// TwinCAT 3 PLC project DAS_A2
// ProgramVersion: 3.1.4020.4
// libraries:
//   Tc2_Standard, * (Beckhoff Automation GmbH)
//   Tc2_System, * (Beckhoff Automation GmbH)
//   Tc3_Module, * (Beckhoff Automation GmbH)
// project tree:
//   DUTs/ ST_PALLET.TcDUT
//   / GlobalTextList.TcGTLO, PlcTask.TcTTO, Visualization Manager.TcVMO (not stored)
//   POUs/ MAIN.TcPOU
//   VISUs/ Visualization.TcVIS

CONFIGURATION DAS_A2
    RESOURCE PLC ON TwinCAT3
        TASK PlcTask(INTERVAL := T#10ms, PRIORITY := 20);
        PROGRAM MAIN WITH PlcTask : MAIN;
    END_RESOURCE
END_CONFIGURATION

// ---- DUTs/ST_PALLET.TcDUT
TYPE ST_PALLET :
STRUCT
	WS1: BOOL;
	WS2: BOOL;
	WS3: BOOL;
	STATE: INT := -1 ;
END_STRUCT
END_TYPE

// ---- POUs/MAIN.TcPOU
PROGRAM MAIN
VAR
	L1: BOOL;   //lock sesnsor1
	L2: BOOL;   //lock sesnsor2
	L3: BOOL;   //lock sesnsor3
	S1: BOOL;   //stopper1 
	S2: BOOL;   //stopper2
	S3: BOOL;   //stopper3
	BA1: BOOL;  //board available1
	BA2: BOOL;  //board available2
	BA3: BOOL;  //board available3
	P1: BOOL;   //presence sesnsor1
	P2: BOOL;   //presence sesnsor2
	P3: BOOL;   //presence sesnsor3
	T1: TON;    //timer for work station1
	T2: TON;    //timer for work station2
	T3: TON;    //timer for work station3
	COUNT_IN: INT;  //number of imported pallets 
	COUNT_OUT: INT;  //number of exported pallets
	PALLETI: ARRAY [1..10] OF ST_PALLET; //each index of this array use for one pallet
	PALLETV: ARRAY[1..10] OF ST_PALLET;  //for saving data of palleti array
	I: INT:=0;  //variable of for loop
	INPUT_PALLET: BOOL; //button for importing pallet to conveyor
	INPUT_PALLET_Pressed: BOOL; // these 3 input pallet used for counting input pallet button just one time in several cycle
	INPUT_PALLET_Released: BOOL;  //
	INPUT_PALLET_PressedBefore: BOOL;  //
	StartStop: BOOL;  //using for start and stop system
	MOTOR: BOOL; //motor of conveyor
	RESET_OUTV1: BOOL;  //exit pallet1 from system
	RESET_OUTV2: BOOL;  //exit pallet2 from system
	RESET_OUTV3: BOOL;  //exit pallet3 from system
	RESET_OUTV4: BOOL;  //exit pallet4 from system
	RESET_OUTV5: BOOL;  //exit pallet5 from system
	RESET_OUTV6: BOOL;  //exit pallet6 from system
	RESET_OUTV7: BOOL;  //exit pallet7 from system
	RESET_OUTV8: BOOL;  //exit pallet8 from system
	RESET_OUTV9: BOOL;  //exit pallet9 from system
	RESET_OUTV10: BOOL;  //exit pallet10 from system
END_VAR

T1(IN:=L1,PT:=T#5S);
T2(IN:=L2,PT:=T#5S);
T3(IN:=L3,PT:=T#5S);

IF INPUT_PALLET_Pressed THEN
	INPUT_PALLET_PressedBefore := TRUE;
ELSIF INPUT_PALLET_Pressed = FALSE AND INPUT_PALLET_PressedBefore THEN
	INPUT_PALLET := TRUE;
	INPUT_PALLET_PressedBefore := FALSE;
END_IF

//START AND INSERT PALLET TO THE SYSTEM AND FOR LOOP IS FOR PREVENTING PROGRAM FROM OVERWRITING DATA OF PALLETS ON PREVIOUS ARRAY INDEXES
	IF StartStop THEN
		MOTOR:=TRUE;
		IF INPUT_PALLET AND (COUNT_IN-COUNT_OUT)<11 THEN
		COUNT_IN:=COUNT_IN +1;
		FOR I:= 1 TO 10 DO
			IF PALLETI[I].STATE = -1 THEN
				PALLETI[I].STATE := 0;
				EXIT;
			END_IF
		END_FOR
		INPUT_PALLET := FALSE;
	END_IF
	
	
	//RESETING OUTPUT MEMORY FOR EACH PALLET
	IF RESET_OUTV1 THEN
			PALLETV[1].WS1:=FALSE;
			PALLETV[1].WS2:=FALSE;
			PALLETV[1].WS3:=FALSE;
			PALLETV[1].STATE:=0;
		END_IF
		IF RESET_OUTV2 THEN
			PALLETV[2].WS1:=FALSE;
			PALLETV[2].WS2:=FALSE;
			PALLETV[2].WS3:=FALSE;
			PALLETV[2].STATE:=0;
		END_IF
		IF RESET_OUTV3 THEN
			PALLETV[3].WS1:=FALSE;
			PALLETV[3].WS2:=FALSE;
			PALLETV[3].WS3:=FALSE;
			PALLETV[3].STATE:=0;
		END_IF
		IF RESET_OUTV4 THEN
			PALLETV[4].WS1:=FALSE;
			PALLETV[4].WS2:=FALSE;
			PALLETV[4].WS3:=FALSE;
			PALLETV[4].STATE:=0;
		END_IF
		IF RESET_OUTV5 THEN
			PALLETV[5].WS1:=FALSE;
			PALLETV[5].WS2:=FALSE;
			PALLETV[5].WS3:=FALSE;
			PALLETV[5].STATE:=0;
		END_IF
		IF RESET_OUTV6 THEN
			PALLETV[6].WS1:=FALSE;
			PALLETV[6].WS2:=FALSE;
			PALLETV[6].WS3:=FALSE;
			PALLETV[6].STATE:=0;
		END_IF
		IF RESET_OUTV7 THEN
			PALLETV[7].WS1:=FALSE;
			PALLETV[7].WS2:=FALSE;
			PALLETV[7].WS3:=FALSE;
			PALLETV[7].STATE:=0;
		END_IF
		IF RESET_OUTV8 THEN
			PALLETV[8].WS1:=FALSE;
			PALLETV[8].WS2:=FALSE;
			PALLETV[8].WS3:=FALSE;
			PALLETV[8].STATE:=0;
		END_IF
		IF RESET_OUTV9 THEN
			PALLETV[9].WS1:=FALSE;
			PALLETV[9].WS2:=FALSE;
			PALLETV[9].WS3:=FALSE;
			PALLETV[9].STATE:=0;
		END_IF
		IF RESET_OUTV10 THEN
			PALLETV[10].WS1:=FALSE;
			PALLETV[10].WS2:=FALSE;
			PALLETV[10].WS3:=FALSE;
			PALLETV[10].STATE:=0;
		END_IF
		
//MAIN FOR LOOP FOR WORKING ON PALLETS		
	FOR I:=1 TO 10 DO
		CASE PALLETI[I].STATE OF        //CHECKING DIFFERENT STATES FOR EACH PALLET
		   -1:
				CONTINUE;
			0:
			IF PALLETI[I].WS1 AND PALLETI[I].WS2 AND PALLETI[I].WS3 THEN
			    PALLETI[I].STATE:=10;
			END_IF	
			IF NOT L1 AND NOT L2 AND NOT L3 THEN
				IF NOT PALLETI[I].WS1 THEN
				PALLETI[I].STATE:=1;
				ELSIF NOT PALLETI[I].WS2 THEN
					PALLETI[I].STATE:=4;
				ELSIF NOT PALLETI[I].WS3 THEN
					PALLETI[I].STATE:=7;
				END_IF
			ELSIF L1 AND NOT L2 AND NOT L3 THEN
				IF NOT PALLETI[I].WS2 THEN
				PALLETI[I].STATE:=4;
				ELSIF NOT PALLETI[I].WS3 THEN
					PALLETI[I].STATE:=7;
				END_IF
			ELSIF L1 AND NOT L2 AND L3 THEN
				IF NOT PALLETI[I].WS2 THEN
				PALLETI[I].STATE:=4;
				END_IF
			ELSIF L1 AND L2 AND NOT L3 THEN
				IF NOT PALLETI[I].WS3 THEN
				PALLETI[I].STATE:=7;
				END_IF
			ELSIF NOT L1 AND L2 AND L3 THEN
				IF NOT PALLETI[I].WS1 THEN
				PALLETI[I].STATE:=1;
				END_IF
			ELSIF NOT L1 AND L2 AND NOT L3 THEN
				IF NOT PALLETI[I].WS3 THEN
				PALLETI[I].STATE:=7;
				END_IF
			ELSIF NOT L1 AND NOT L2 AND L3 THEN
				IF NOT PALLETI[I].WS1 THEN
					PALLETI[I].STATE:=1;
				ELSIF NOT PALLETI[I].WS2 THEN
					PALLETI[I].STATE:=4;
				END_IF
			END_IF
		
			1:  //WORK STATION1 WORKS ON PALLET UP TO STATE3
			IF PALLETI[I].WS1 AND PALLETI[I].WS2 AND PALLETI[I].WS3 THEN
			    PALLETI[I].STATE:=10;
			ELSIF NOT PALLETI[I].WS1 THEN
				IF NOT L1 AND P1 THEN
				BA1:=TRUE;
                S1:=TRUE;
				PALLETI[I].STATE:=2;
			    END_IF
			END_IF
			
			2:
			IF L1 THEN
				T1(IN:=L1,PT:=T#5S);
			    BA1:=FALSE;
			    S1:=FALSE;
				IF T1.Q THEN
					PALLETI[I].STATE:=3;
				END_IF
			END_IF
			
            3:
			IF NOT L1 THEN
				PALLETI[I].WS1:=1;
				IF PALLETI[I].WS1 AND PALLETI[I].WS2 AND PALLETI[I].WS3 THEN
			    PALLETI[I].STATE:=10;
				END_IF
				PALLETI[I].STATE:=0;
			END_IF

			4:   //WORK STATION2 WORKS ON PALLET UP TO STATE7
			IF PALLETI[I].WS1 AND PALLETI[I].WS2 AND PALLETI[I].WS3 THEN
			    PALLETI[I].STATE:=10;
			ELSIF NOT PALLETI[I].WS2 THEN
				IF NOT L2 AND P2 THEN
				BA2:=TRUE;
				S2:=TRUE;
				PALLETI[I].STATE:=5;
			    END_IF
			END_IF
			
            5:
			IF L2 THEN
				BA2:=FALSE;
			    S2:=FALSE;
				IF T2.Q THEN
					PALLETI[I].STATE:=6;
			    END_IF
			END_IF
			
			6:
			IF NOT L2 THEN
				PALLETI[I].WS2:=1;
				IF PALLETI[I].WS1 AND PALLETI[I].WS2 AND PALLETI[I].WS3 THEN
			    PALLETI[I].STATE:=10;
				END_IF
				PALLETI[I].STATE:=0;
			END_IF
			
			7:   //WORK STATION3 WORKS ON PALLET UP TO STATE9
			IF PALLETI[I].WS1 AND PALLETI[I].WS2 AND PALLETI[I].WS3 THEN
			    PALLETI[I].STATE:=10;
			ELSIF NOT PALLETI[I].WS3 THEN
				IF NOT L3 AND P3 THEN
				BA3:=TRUE;
				S3:=TRUE;
				PALLETI[I].STATE:=8;
			    END_IF
			END_IF
			
			8:
			IF L3 THEN
				BA3:=FALSE;
			    S3:=FALSE;
			    IF T3.Q THEN
					PALLETI[I].STATE:=9;
				END_IF
			END_IF
			
			9:
			IF NOT L3 THEN
				PALLETI[I].WS3:=1;
				IF PALLETI[I].WS1 AND PALLETI[I].WS2 AND PALLETI[I].WS3 THEN
			    PALLETI[I].STATE:=10;
				END_IF
				PALLETI[I].STATE:=0;
			END_IF
			
			10:    //TRANSFERING DATA OF PALLETI TO PALLETV AND RESET THE PALLET AND TURN IT BACK
				
				IF  PALLETI[I].WS1 AND PALLETI[I].WS2 AND PALLETI[I].WS3 THEN
					PALLETV[I].WS1:=PALLETI[I].WS1;
					PALLETV[I].WS2:=PALLETI[I].WS2;
					PALLETV[I].WS3:=PALLETI[I].WS3;
					PALLETV[I].STATE:=PALLETI[I].STATE;
			
				
				END_IF
				PALLETI[I].WS1:=FALSE;
				PALLETI[I].WS2:=FALSE;
				PALLETI[I].WS3:=FALSE;
				PALLETI[I].STATE:=-1;
				COUNT_OUT:=COUNT_OUT+1;
		
		END_CASE
	END_FOR
	ELSE 
		MOTOR:=FALSE;
END_IF

END_PROGRAM

// ---- GlobalTextList.TcGTLO
TEXTLIST GlobalTextList
  10 = 'BA1'
  9 = 'BA2'
  11 = 'BA3'
  41 = 'EXIT PALLET1'
  50 = 'EXIT PALLET10'
  42 = 'EXIT PALLET2'
  43 = 'EXIT PALLET3'
  44 = 'EXIT PALLET4'
  45 = 'EXIT PALLET5'
  46 = 'EXIT PALLET6'
  47 = 'EXIT PALLET7'
  48 = 'EXIT PALLET8'
  49 = 'EXIT PALLET9'
  18 = 'Input Pallet'
  3 = 'L1'
  4 = 'L2'
  5 = 'L3'
  15 = 'Motor'
  6 = 'P1'
  7 = 'P2'
  8 = 'P3'
  19 = 'Pallet 1'
  28 = 'Pallet 10'
  20 = 'Pallet 2'
  21 = 'Pallet 3'
  22 = 'Pallet 4'
  23 = 'Pallet 5'
  24 = 'Pallet 6'
  25 = 'Pallet 7'
  26 = 'Pallet 8'
  27 = 'Pallet 9'
  31 = 'R'
  30 = 'RESET PALLET1'
  40 = 'RESET PALLET10'
  32 = 'RESET PALLET2'
  33 = 'RESET PALLET3'
  34 = 'RESET PALLET4'
  35 = 'RESET PALLET5'
  36 = 'RESET PALLET6'
  37 = 'RESET PALLET7'
  38 = 'RESET PALLET8'
  39 = 'RESET PALLET9'
  17 = 'Start'
  29 = 'StartStop'
  16 = 'Stop'
  12 = 'Stopper1'
  13 = 'Stopper2'
  14 = 'Stopper3'
  1 = 'WS1'
  2 = 'WS2'
  0 = 'WS3'
END_TEXTLIST

// ---- VISUs/Visualization.TcVIS
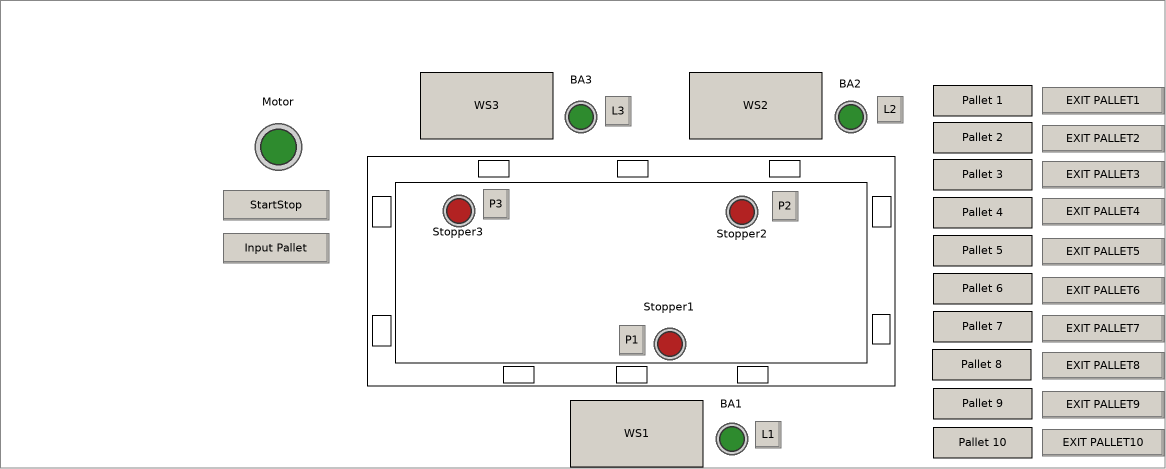
VISUALIZATION Visualization  // 1166x469
    RoundedRectangle (367,156 528x230)
    RoundedRectangle (395,182 472x181)
    Rectangle (570,400 133x67), "WS1", colour toggle: MAIN.T1.Q
    Rectangle (420,72 133x67), "WS3", colour toggle: MAIN.T3.Q
    Rectangle (689,72 133x67), "WS2", colour toggle: MAIN.T2.Q
    Button (755,421 26x27), "L1", text variable: MAIN.L1, colour toggle: MAIN.L1
        toggle MAIN.L1
    Button (605,96 26x30), "L3", text variable: MAIN.L3, colour toggle: MAIN.L3
        toggle MAIN.L3
    Button (483,189 26x30), "P3"
        tap MAIN.P3
    Button (772,191 26x30), "P2"
        tap MAIN.P2
    Button (619,325 26x30), "P1"
        tap MAIN.P1
    Lamp1 (832,94 38x46), tooltip "BA2", variable: MAIN.BA2, style: Lamp-Lamp1-Green
    Label (775,69 150x30), "BA2"
    Lamp1 (562,94 38x46), variable: MAIN.BA3, style: Lamp-Lamp1-Green
    Lamp1 (713,416 38x46), variable: MAIN.BA1, style: Lamp-Lamp1-Green
    Label (506,63 150x34), "BA3"
    Label (656,389 150x30), "BA1"
    Lamp1 (723,189 38x46), variable: MAIN.S2, style: Lamp-Lamp1-Red
    Lamp1 (440,188 38x46), variable: MAIN.S3, style: Lamp-Lamp1-Red
    Lamp1 (651,321 38x46), variable: MAIN.S1, style: Lamp-Lamp1-Red
    Label (594,292 150x30), "Stopper1"
    Label (383,217 150x30), "Stopper3"
    Label (667,219 150x30), "Stopper2"
    Rectangle (503,366 31x17)
    Lamp1 (251,115 55x64), variable: MAIN.MOTOR, style: Lamp-Lamp1-Green
    Label (203,87 150x30), "Motor"
    Button (223,190 106x30), "StartStop"
        toggle MAIN.StartStop
    Button (223,233 106x30), "Input Pallet"
        tap MAIN.INPUT_PALLET_Pressed
    Button (877,96 26x27), "L2", text variable: MAIN.L2, colour toggle: MAIN.L2
        toggle MAIN.L2
    Rectangle (933,85 99x31), "Pallet 1", colour toggle: MAIN.PALLETV[1].WS1
    Rectangle (372,315 19x31)
    Rectangle (617,160 31x17)
    Rectangle (769,160 31x17), invisible if: MAIN.L2
    Rectangle (478,160 31x17), invisible if: MAIN.L3
    Rectangle (737,366 31x17)
    Rectangle (616,366 31x17), invisible if: MAIN.L1
    Rectangle (872,314 18x30)
    Rectangle (872,196 19x31)
    Rectangle (372,196 19x31)
    Rectangle (933,122 99x31), "Pallet 2", colour toggle: MAIN.PALLETV[2].WS1
    Rectangle (933,159 99x31), "Pallet 3", colour toggle: MAIN.PALLETV[3].WS1
    Rectangle (933,197 99x31), "Pallet 4", colour toggle: MAIN.PALLETV[4].WS1
    Rectangle (933,235 99x31), "Pallet 5", colour toggle: MAIN.PALLETV[5].WS1
    Rectangle (933,273 99x31), "Pallet 6", colour toggle: MAIN.PALLETV[6].WS1
    Rectangle (933,311 99x31), "Pallet 7", colour toggle: MAIN.PALLETV[7].WS1
    Rectangle (932,349 99x31), "Pallet 8", colour toggle: MAIN.PALLETV[8].WS1
    Rectangle (933,388 99x31), "Pallet 9", colour toggle: MAIN.PALLETV[9].WS1
    Rectangle (933,427 99x31), "Pallet 10", colour toggle: MAIN.PALLETV[10].WS1
    Button (1042,87 122x27), "EXIT PALLET1"
        tap MAIN.RESET_OUTV1
    Button (1042,198 122x27), "EXIT PALLET4"
        tap MAIN.RESET_OUTV4
    Button (1042,238 122x27), "EXIT PALLET5"
        tap MAIN.RESET_OUTV5
    Button (1042,277 122x27), "EXIT PALLET6"
        tap MAIN.RESET_OUTV6
    Button (1042,315 122x27), "EXIT PALLET7"
        tap MAIN.RESET_OUTV7
    Button (1042,352 122x27), "EXIT PALLET8"
        tap MAIN.RESET_OUTV8
    Button (1042,391 122x27), "EXIT PALLET9"
        tap MAIN.RESET_OUTV9
    Button (1042,429 122x27), "EXIT PALLET10"
        tap MAIN.RESET_OUTV10
    Button (1042,161 122x27), "EXIT PALLET3"
        tap MAIN.RESET_OUTV3
    Button (1042,125 122x27), "EXIT PALLET2"
        tap MAIN.RESET_OUTV2
END_VISUALIZATION
